(* IEC 61131-3 sources: AXOpen/src/sdk-ax/ctrl/src, 1 file *)

(* ---- class1.st ---- *)
NAMESPACE MyNamespace
    CLASS class1
        VAR PUBLIC
            Hello : STRING;
        END_VAR

    END_CLASS

END_NAMESPACE
